PROGRAM MAIN
VAR
END_VAR

fbAct1();

END_PROGRAM

(* stored: Version 1.1.0.1, ProductVersion 3.1.4020.6
   POU MAIN: Id {cbc2c2b7-1a3a-4853-bcb5-af497b57f77a}, SpecialFunc None *)
